Yaskawa INFORM job: ariel_test_29_12_2022.JBI

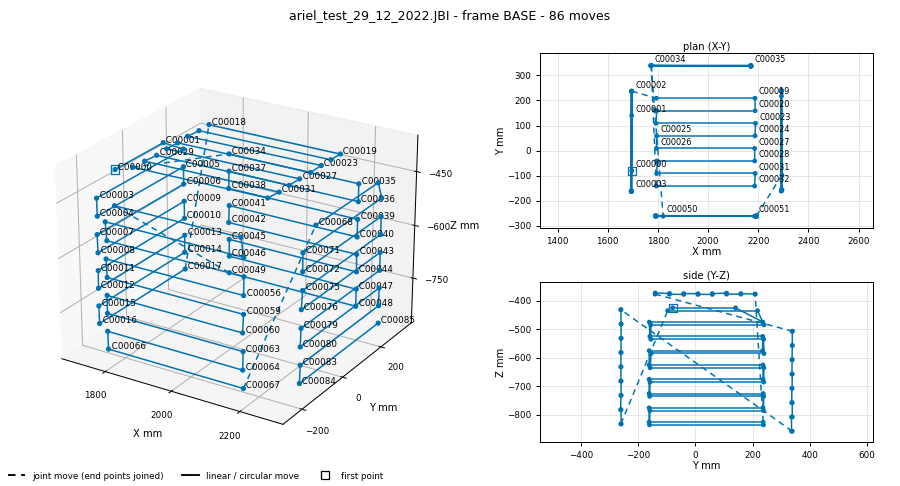
[picture p0: tool path of ariel_test_29_12_2022.JBI in frame BASE, 86 of 86 moves have a stored position in this frame; points joined in program order, loops and branches not executed]
/JOB
//NAME test1
//POS
///NPOS 86,0,0,0,0,0
///TOOL 0
///POSTYPE BASE
///RECTAN
///RCONF 1,0,0,0,0,0,0,0,0,0,0,0,0,0,0,0,0,0,0,0,0,0,0,0
C00000=1696.132000,-80.047400,-425.128800,-2.796034,72.857313,-92.928025
C00001=1695.649900,140.027500,-425.128800,-7.866711,71.298868,-98.296639
C00002=1695.009700,236.007500,-475.128800,112.293998,77.773291,21.835422
C00003=1694.894300,-161.509200,-475.128800,-88.057884,81.491787,-178.075283
C00004=1694.500400,-159.876400,-525.128800,-78.924936,82.712187,-169.011090
C00005=1694.957700,235.269700,-525.128800,103.854330,80.552136,13.676503
C00006=1695.172400,234.870300,-575.128800,89.117855,76.604457,-0.859437
C00007=1694.072400,-162.036300,-575.128800,-85.708757,79.755725,-175.777722
C00008=1695.266200,-162.303200,-625.128800,-93.965078,72.880232,176.207440
C00009=1695.465900,236.123700,-625.128800,87.238554,69.471133,-2.589769
C00010=1695.422700,236.644700,-675.128800,91.163315,69.247679,1.088620
C00011=1694.457900,-162.352100,-675.128800,-85.937940,81.468869,-175.978257
C00012=1693.613400,-162.296700,-725.128800,-77.292007,71.866096,-167.905282
C00013=1695.359600,236.966000,-725.128800,93.357743,70.594130,3.168457
C00014=1695.305600,236.328100,-775.128800,92.916566,74.123550,2.801764
C00015=1693.299800,-162.503900,-775.128800,-70.983741,81.245415,-161.190217
C00016=1694.079700,-162.510900,-825.128800,-105.768009,75.653347,164.696718
C00017=1695.793500,236.889300,-825.128800,96.268369,73.447460,6.010327
C00018=1793.675300,208.803900,-377.180700,-3.976327,1.157375,-90.000210
C00019=2187.017900,208.803900,-377.015400,0.372423,-2.698631,-90.000210
C00020=2187.698900,158.803900,-375.418500,0.853707,-9.201702,-90.000210
C00021=1795.170400,158.803900,-377.409600,0.882355,-3.248671,-90.000210
C00022=1792.375400,108.803900,-377.337500,-8.863657,1.902220,-90.000210
C00023=2189.165300,108.803900,-373.615200,-4.858682,5.196727,-90.000210
C00024=2187.408900,58.803900,-375.476400,-0.670361,-6.886953,-90.000210
C00025=1795.003900,58.803900,-378.201600,-2.904896,-6.755172,-90.000210
C00026=1794.543100,8.803900,-378.074400,-0.080214,2.297561,-90.000210
C00027=2185.685100,8.803900,-375.544700,-0.899544,8.640204,-90.000210
C00028=2185.880000,-41.196100,-375.195400,-1.117268,8.600097,-90.000210
C00029=1797.809600,-41.196100,-378.167200,7.883899,-5.792603,-90.000210
C00030=1795.305000,-91.196100,-377.541600,1.054242,7.110406,-90.000210
C00031=2187.800700,-91.196100,-374.817700,-0.160428,-3.116890,-90.000210
C00032=2185.655400,-141.196100,-373.016400,9.625691,-3.042406,-90.000210
C00033=1793.794000,-141.196100,-377.211700,-1.804817,16.667342,-90.000210
C00034=1773.422800,338.858700,-507.069300,91.827946,12.026384,0.383882
C00035=2170.526400,339.076800,-507.069300,94.830245,-6.892682,-0.578687
C00036=2170.470000,338.721700,-557.069300,90.028858,-18.707072,-0.011459
C00037=1772.765600,338.845000,-557.069300,91.833675,19.767044,0.618794
C00038=1772.113800,338.178100,-607.069300,87.742757,19.383162,-0.750575
C00039=2169.918900,338.249700,-607.069300,90.865377,-18.729990,-0.280749
C00040=2169.846800,337.617600,-657.069300,91.742002,-19.933202,-0.595876
C00041=1773.408600,338.699100,-657.069300,91.191963,19.411810,0.395341
C00042=1771.966000,338.269300,-707.069300,91.770650,17.778880,0.538580
C00043=2169.887200,337.437200,-707.069300,91.123208,-14.054655,-0.275020
C00044=2170.816100,336.900000,-757.069300,92.177450,-3.495043,-0.131780
C00045=1773.075800,338.832900,-757.069300,92.515495,19.308678,0.830789
C00046=1773.335100,338.792700,-807.069300,92.595709,17.813258,0.796411
C00047=2171.727500,336.247000,-807.069300,89.547574,-16.105844,0.126051
C00048=2171.220400,336.110800,-857.069300,92.859270,-14.661990,-0.727656
C00049=1773.221800,338.627300,-857.069300,89.243906,16.420970,-0.211994
C00050=1820.971900,-261.541800,-431.614400,-77.561297,0.315127,-179.931666
C00051=2184.952000,-261.044500,-431.614400,-83.296604,2.647065,-179.691024
C00052=2192.839600,-260.681700,-481.614400,-88.550627,-12.226919,179.691024
C00053=1791.152000,-260.567100,-481.614400,-101.636983,48.323260,171.257085
C00054=1794.425600,-260.324700,-531.614400,-90.561709,7.024463,179.931666
C00055=2193.314000,-261.064500,-531.614400,-93.839028,-17.480942,-178.843046
C00056=2192.341900,-260.734400,-581.614400,-90.372633,-8.130271,-179.948855
C00057=1791.071900,-261.005300,-581.614400,-89.593410,12.547776,-179.908748
C00058=1793.131800,-261.280300,-631.614400,-86.510897,12.043573,-179.272765
C00059=2192.209400,-260.873200,-631.614400,-90.172098,-14.931280,-179.954584
C00060=2189.954000,-261.359600,-681.614400,-90.573168,-4.503448,-179.954584
C00061=1791.050300,-260.611400,-681.614400,-91.042994,-1.621471,-179.971773
C00062=1790.464400,-260.376300,-731.614400,-86.149934,10.032491,-179.330060
C00063=2191.354100,-261.246600,-731.614400,-90.727867,-16.014170,-179.799886
C00064=2190.798500,-262.036100,-781.614400,-90.716408,-16.478266,-179.799886
C00065=1790.058300,-260.739400,-781.614400,-94.480740,10.891928,179.152443
C00066=1790.686400,-260.189100,-831.614400,-89.347039,15.412565,-179.828534
C00067=2192.318900,-261.278300,-831.614400,-83.090339,-16.231894,178.058094
C00068=2294.292800,-97.327000,-435.033100,7.689094,-78.890559,82.167877
C00069=2292.553200,217.265700,-435.033100,5.821251,-50.448934,82.471545
C00070=2291.804400,239.786900,-485.033100,116.018224,-82.334035,-25.811749
C00071=2294.201800,-156.615000,-485.033100,-92.028481,-82.391331,-177.989339
C00072=2293.933400,-156.359200,-535.033100,-113.915469,-85.233202,-156.159647
C00073=2292.245400,238.334100,-535.033100,88.934509,-85.559788,1.065701
C00074=2291.848800,239.682800,-585.033100,87.937562,-72.817206,1.965245
C00075=2293.799300,-155.333200,-585.033100,-84.981100,-84.625866,175.004229
C00076=2292.833100,-158.703500,-635.033100,-83.542976,-73.361516,173.812477
C00077=2291.947400,239.284200,-635.033100,88.206853,-75.429894,1.736062
C00078=2292.084100,238.852100,-685.033100,87.387523,-69.998254,2.452259
C00079=2292.973900,-159.159300,-685.033100,-37.179231,-85.112880,127.276845
C00080=2292.114000,-160.465100,-735.033100,-81.921506,-79.085364,172.064955
C00081=2291.977800,238.820300,-735.033100,91.656058,-71.528051,-1.569904
C00082=2292.135300,237.997300,-785.033100,89.306932,-73.613618,0.664631
C00083=2292.381400,-159.627800,-785.033100,-111.417373,-80.208362,-158.869737
C00084=2291.307500,-160.899900,-835.033100,-80.534948,-71.556699,171.016443
C00085=2292.416200,237.973300,-835.033100,103.670983,-73.997499,-13.160841
//INST
///DATE 2022/12/29 10:08
///ATTR SC,RW,RJ
////FRAME BASE
///GROUP1 RB1
NOP
MOVJ C00000 VJ=50.00
MOVL C00001 V=350.0
MOVL C00002 V=350.0
MOVL C00003 V=350.0
MOVL C00004 V=350.0
MOVL C00005 V=350.0
MOVL C00006 V=350.0
MOVL C00007 V=350.0
MOVL C00008 V=350.0
MOVL C00009 V=350.0
MOVL C00010 V=350.0
MOVL C00011 V=350.0
MOVL C00012 V=350.0
MOVL C00013 V=350.0
MOVL C00014 V=350.0
MOVL C00015 V=350.0
MOVL C00016 V=350.0
MOVL C00017 V=350.0
MOVJ C00018 VJ=50.00
MOVL C00019 V=350.0
MOVL C00020 V=350.0
MOVL C00021 V=350.0
MOVL C00022 V=350.0
MOVL C00023 V=350.0
MOVL C00024 V=350.0
MOVL C00025 V=350.0
MOVL C00026 V=350.0
MOVL C00027 V=350.0
MOVL C00028 V=350.0
MOVL C00029 V=350.0
MOVL C00030 V=350.0
MOVL C00031 V=350.0
MOVL C00032 V=350.0
MOVL C00033 V=350.0
MOVJ C00034 VJ=50.00
MOVL C00035 V=350.0
MOVL C00036 V=350.0
MOVL C00037 V=350.0
MOVL C00038 V=350.0
MOVL C00039 V=350.0
MOVL C00040 V=350.0
MOVL C00041 V=350.0
MOVL C00042 V=350.0
MOVL C00043 V=350.0
MOVL C00044 V=350.0
MOVL C00045 V=350.0
MOVL C00046 V=350.0
MOVL C00047 V=350.0
MOVL C00048 V=350.0
MOVL C00049 V=350.0
MOVJ C00050 VJ=50.00
MOVL C00051 V=350.0
MOVL C00052 V=350.0
MOVL C00053 V=350.0
MOVL C00054 V=350.0
MOVL C00055 V=350.0
MOVL C00056 V=350.0
MOVL C00057 V=350.0
MOVL C00058 V=350.0
MOVL C00059 V=350.0
MOVL C00060 V=350.0
MOVL C00061 V=350.0
MOVL C00062 V=350.0
MOVL C00063 V=350.0
MOVL C00064 V=350.0
MOVL C00065 V=350.0
MOVL C00066 V=350.0
MOVL C00067 V=350.0
MOVJ C00068 VJ=50.00
MOVL C00069 V=350.0
MOVL C00070 V=350.0
MOVL C00071 V=350.0
MOVL C00072 V=350.0
MOVL C00073 V=350.0
MOVL C00074 V=350.0
MOVL C00075 V=350.0
MOVL C00076 V=350.0
MOVL C00077 V=350.0
MOVL C00078 V=350.0
MOVL C00079 V=350.0
MOVL C00080 V=350.0
MOVL C00081 V=350.0
MOVL C00082 V=350.0
MOVL C00083 V=350.0
MOVL C00084 V=350.0
MOVL C00085 V=350.0
END
